FUNCTION GetResourceFromCommand : STRING
VAR_INPUT
	Command: STRING;
END_VAR
VAR
	sReturn : STRING;
END_VAR

sReturn := LEFT ( Command , FIND(Command,'_') - 1);
GetResourceFromCommand := sReturn;

END_FUNCTION

(* stored: Version 1.1.0.1, ProductVersion 3.1.4020.3
   POU GetResourceFromCommand: Id {1127ab92-b28c-4365-9ea6-613002fde49d}, SpecialFunc None *)
